Staubli VAL3: SHL.pgx

public program SHL(num x_shift, num& x_value[])
// shift num value to left
begin
  if bDebug
    putln("SHL()")
  endIf
  x_value=roundDown(x_value)*exp(roundDown(x_shift)*ln(2))
end
